FUNCTION_BLOCK L1_L1CFB (* Composite Function Block Type *)
  (* Standard: 61499-2; Description: This block encapsulates all the step-nc feature-FB translating blocks. These translate a feature of the process plan into a set of consecutive orders that a CNC can understand and execute. *)
  (* Version 0.0, 2015-03-18, EQUEROL, UJI *)
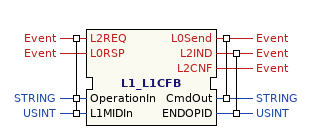
  EVENT_INPUT
    L2REQ WITH OperationIn, L1MIDIn; (* Request multicast send to all blocks in layer 1 *)
    L0RSP; (* Cmd reception confirmation *)
  END_EVENT
  EVENT_OUTPUT
    L0Send WITH CmdOut; (* Execution Confirmation *)
    L2IND WITH ENDOPID; (* Communication Failure indication *)
    L2CNF; (* Confirmation of Requested Service *)
  END_EVENT
  VAR_INPUT
    OperationIn : STRING; (* Serialized operation *)
    L1MIDIn : USINT; (* Layer 1 multicast identifier *)
  END_VAR
  VAR_OUTPUT
    CmdOut : STRING; (* Command to be sent to the machine *)
    ENDOPID : USINT; (* Indicate upper layer that operation failed *)
  END_VAR
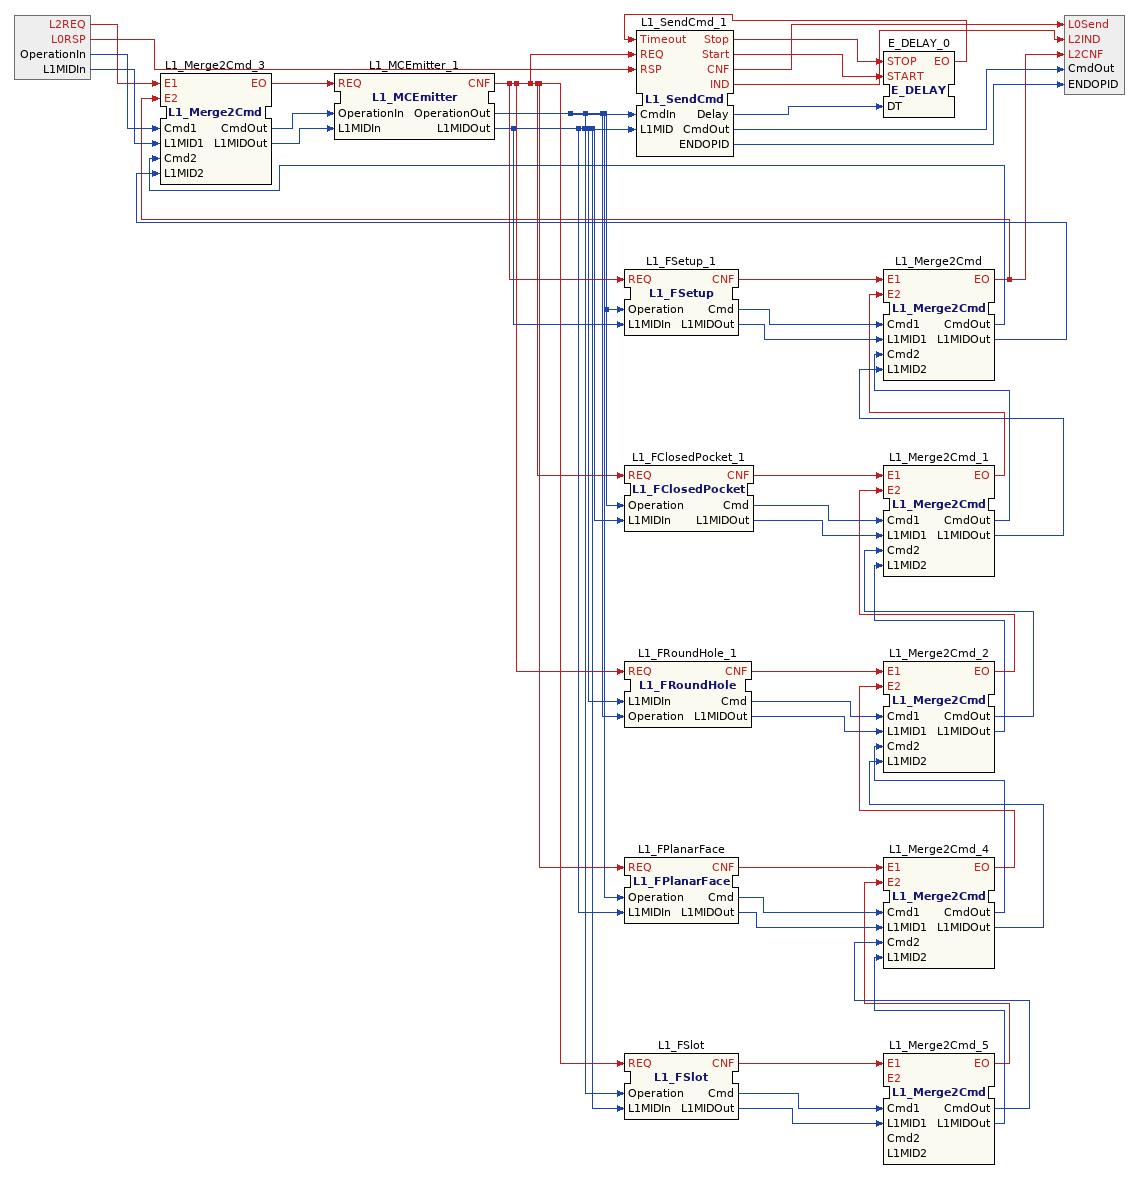
  FBS
    E_DELAY_0 : E_DELAY;
    L1_MCEmitter_1 : L1_MCEmitter;
    L1_FSetup_1 : L1_FSetup;
    L1_SendCmd_1 : L1_SendCmd;
    L1_FClosedPocket_1 : L1_FClosedPocket;
    L1_FRoundHole_1 : L1_FRoundHole;
    L1_Merge2Cmd : L1_Merge2Cmd;
    L1_Merge2Cmd_1 : L1_Merge2Cmd;
    L1_Merge2Cmd_2 : L1_Merge2Cmd;
    L1_Merge2Cmd_3 : L1_Merge2Cmd;
    L1_Merge2Cmd_4 : L1_Merge2Cmd;
    L1_FPlanarFace : L1_FPlanarFace;
    L1_FSlot : L1_FSlot;
    L1_Merge2Cmd_5 : L1_Merge2Cmd;
  END_FBS
  EVENT_CONNECTIONS
    L1_MCEmitter_1.CNF TO L1_FSetup_1.REQ;
    L1_MCEmitter_1.CNF TO L1_FRoundHole_1.REQ;
    E_DELAY_0.EO TO L1_SendCmd_1.Timeout;
    L1_MCEmitter_1.CNF TO L1_SendCmd_1.REQ;
    L1_MCEmitter_1.CNF TO L1_FClosedPocket_1.REQ;
    L1_SendCmd_1.Stop TO E_DELAY_0.STOP;
    L1_SendCmd_1.Start TO E_DELAY_0.START;
    L0RSP TO L1_SendCmd_1.RSP;
    L1_SendCmd_1.CNF TO L0Send;
    L1_SendCmd_1.IND TO L2IND;
    L1_FSetup_1.CNF TO L1_Merge2Cmd.E1;
    L1_Merge2Cmd_1.EO TO L1_Merge2Cmd.E2;
    L1_FClosedPocket_1.CNF TO L1_Merge2Cmd_1.E1;
    L1_Merge2Cmd_2.EO TO L1_Merge2Cmd_1.E2;
    L1_FRoundHole_1.CNF TO L1_Merge2Cmd_2.E1;
    L1_Merge2Cmd.EO TO L2CNF;
    L2REQ TO L1_Merge2Cmd_3.E1;
    L1_Merge2Cmd_3.EO TO L1_MCEmitter_1.REQ;
    L1_Merge2Cmd.EO TO L1_Merge2Cmd_3.E2;
    L1_Merge2Cmd_4.EO TO L1_Merge2Cmd_2.E2;
    L1_MCEmitter_1.CNF TO L1_FPlanarFace.REQ;
    L1_FPlanarFace.CNF TO L1_Merge2Cmd_4.E1;
    L1_FSlot.CNF TO L1_Merge2Cmd_5.E1;
    L1_MCEmitter_1.CNF TO L1_FSlot.REQ;
    L1_Merge2Cmd_5.EO TO L1_Merge2Cmd_4.E2;
  END_CONNECTIONS
  DATA_CONNECTIONS
    L1_MCEmitter_1.OperationOut TO L1_FSetup_1.Operation;
    L1_MCEmitter_1.OperationOut TO L1_SendCmd_1.CmdIn;
    L1_MCEmitter_1.L1MIDOut TO L1_FRoundHole_1.L1MIDIn;
    L1_MCEmitter_1.L1MIDOut TO L1_SendCmd_1.L1MID;
    L1_MCEmitter_1.OperationOut TO L1_FRoundHole_1.Operation;
    L1_SendCmd_1.Delay TO E_DELAY_0.DT;
    L1_MCEmitter_1.L1MIDOut TO L1_FClosedPocket_1.L1MIDIn;
    L1_MCEmitter_1.L1MIDOut TO L1_FSetup_1.L1MIDIn;
    L1_MCEmitter_1.OperationOut TO L1_FClosedPocket_1.Operation;
    L1_SendCmd_1.CmdOut TO CmdOut;
    L1_SendCmd_1.ENDOPID TO ENDOPID;
    L1_Merge2Cmd_1.CmdOut TO L1_Merge2Cmd.Cmd2;
    L1_Merge2Cmd_1.L1MIDOut TO L1_Merge2Cmd.L1MID2;
    L1_FSetup_1.Cmd TO L1_Merge2Cmd.Cmd1;
    L1_FSetup_1.L1MIDOut TO L1_Merge2Cmd.L1MID1;
    L1_FClosedPocket_1.Cmd TO L1_Merge2Cmd_1.Cmd1;
    L1_FClosedPocket_1.L1MIDOut TO L1_Merge2Cmd_1.L1MID1;
    L1_Merge2Cmd_2.CmdOut TO L1_Merge2Cmd_1.Cmd2;
    L1_Merge2Cmd_2.L1MIDOut TO L1_Merge2Cmd_1.L1MID2;
    L1_FRoundHole_1.Cmd TO L1_Merge2Cmd_2.Cmd1;
    L1_FRoundHole_1.L1MIDOut TO L1_Merge2Cmd_2.L1MID1;
    OperationIn TO L1_Merge2Cmd_3.Cmd1;
    L1MIDIn TO L1_Merge2Cmd_3.L1MID1;
    L1_Merge2Cmd.CmdOut TO L1_Merge2Cmd_3.Cmd2;
    L1_Merge2Cmd.L1MIDOut TO L1_Merge2Cmd_3.L1MID2;
    L1_Merge2Cmd_3.CmdOut TO L1_MCEmitter_1.OperationIn;
    L1_Merge2Cmd_3.L1MIDOut TO L1_MCEmitter_1.L1MIDIn;
    L1_Merge2Cmd_4.CmdOut TO L1_Merge2Cmd_2.Cmd2;
    L1_Merge2Cmd_4.L1MIDOut TO L1_Merge2Cmd_2.L1MID2;
    L1_MCEmitter_1.OperationOut TO L1_FPlanarFace.Operation;
    L1_FPlanarFace.Cmd TO L1_Merge2Cmd_4.Cmd1;
    L1_FPlanarFace.L1MIDOut TO L1_Merge2Cmd_4.L1MID1;
    L1_MCEmitter_1.L1MIDOut TO L1_FPlanarFace.L1MIDIn;
    L1_MCEmitter_1.OperationOut TO L1_FSlot.Operation;
    L1_MCEmitter_1.L1MIDOut TO L1_FSlot.L1MIDIn;
    L1_FSlot.Cmd TO L1_Merge2Cmd_5.Cmd1;
    L1_FSlot.L1MIDOut TO L1_Merge2Cmd_5.L1MID1;
    L1_Merge2Cmd_5.CmdOut TO L1_Merge2Cmd_4.Cmd2;
    L1_Merge2Cmd_5.L1MIDOut TO L1_Merge2Cmd_4.L1MID2;
  END_CONNECTIONS
END_FUNCTION_BLOCK
